Universal Robots PolyScope program: test_2.urp

Program test_2 (installation=default directory=/home/ur/ursim-current/programs createdIn=5.8.0.10253 lastSavedIn=5.8.0.10253 robotSerialNumber=20195599999)
Calibrated DH parameters: a=[0, -0.425, -0.3922, 0, 0, 0]; d=[0.1625, 0, 0, 0.1333, 0.0997, 0.0996]; alpha=[1.570796, 0, 0, 1.570796, -1.570796, 0]; deltaTheta=[0, 0, 0, 0, 0, 0]
Robot Program (runOnlyOnce=false)
  Set DigitalOutput pin=digital_out[0]; digitalValue=0
  Wait Sleep waitTime=1
  Set DigitalOutput pin=digital_out[0]; digitalValue=1
  MoveJ speed 60 deg/s, acceleration 80 deg/s^2 (useActiveTCP=true) feature=Base
    Waypoint Waypoint_1: TCP in base x=502.012 y=-130.88 z=120.73 mm, rx=-2.0212 ry=1.9495 rz=-0.4007 rad; joints [0, -120, -126.223, 0, 91.392, -1.776] deg
  MoveJ speed 60 deg/s, acceleration 80 deg/s^2 (useActiveTCP=true) feature=Base
    Waypoint Waypoint_2: TCP in base x=508.171 y=-130.88 z=969.916 mm, rx=-0.156 ry=1.5642 rz=-0.118 rad; joints [0, -120, 0, -60, 91.392, 80] deg
Thread Thread_1 (runOnlyOnce=false)
  Wait Condition expression=read_input_boolean_register(65)
  Halt
